(* IEC 61131-3 sources: hayabusa-infrastructure-templates/Ansible/SCADA & PLC/programs, 1 file *)

(* ---- example.st ---- *)
PROGRAM Example
VAR
    start_button : BOOL;
    motor_output : BOOL;
END_VAR

motor_output := start_button;
END_PROGRAM
